// Mitsubishi GX Works2 project: test   PLC: Q03UDV

PROGRAM MAIN
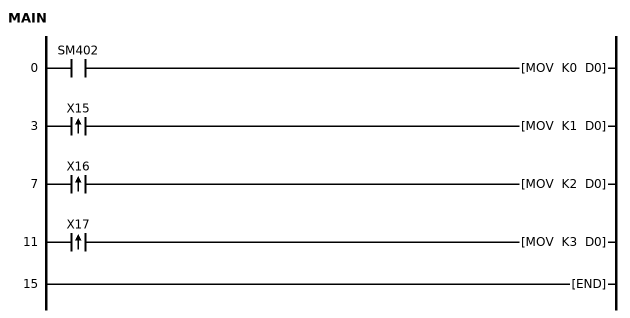
0     LD      SM402
      MOV     K0 D0
3     LDP     X15
      MOV     K1 D0
7     LDP     X16
      MOV     K2 D0
11    LDP     X17
      MOV     K3 D0
15    END
END_PROGRAM

// device comments not shown above
X0  ; 공급 후진
X1  ; 공급 전진
X2  ; 분배 후진
X3  ; 분배 전진
X4  ; 가공 상승
X5  ; 가공 하강
Y20  ; 공급+
Y21  ; 공급-
Y22  ; 분배+
Y23  ; 분배-
Y24  ; 가공+/-
M10  ; 공급 동작
M11  ; 분배 동작
M12  ; 가공 동작
M100  ; 초기화
M101  ; 초기화
M200  ; 코멘트
